// TIA Portal V17 export
// export: Created 2022-03-12T16:05:07.905036Z, ExportSetting WithDefaults, DisplayName Totally Integrated Automation Portal, DisplayVersion V17, DisplayName TIA Portal Openness, DisplayVersion V17, DisplayName TIA Portal Version Control Interface, DisplayVersion V17, DisplayName STEP 7 Professional, DisplayVersion V17, DisplayName STEP 7 Safety, DisplayVersion V17, DisplayName WinCC Advanced / Unified PC, DisplayVersion V17
ORGANIZATION_BLOCK "Main"   // OB1, LAD, ProgramCycle
TITLE = Main
{ S7_Optimized_Access := 'TRUE' }
AUTHOR : tech.team.motioncontrol@siemens.com
FAMILY : CPG
VERSION : 1.0
// Support: tech.team.motioncontrol@siemens.com
// Fax: +49 (0) 9131/98-1297
// stored: AutoNumber true, IsIECCheckEnabled false, SetENOAutomatically false
   VAR_INPUT
      Initial_Call : Bool;   // Initial call of this OB
      Remanence : Bool;   // =True, if remanent data are available
   END_VAR
   VAR_TEMP   // added for the SCL form of the ladder/FBD networks
      _w1 : Bool;
   END_VAR
BEGIN

REGION Network 1: Factory IO PLCSIM Communication
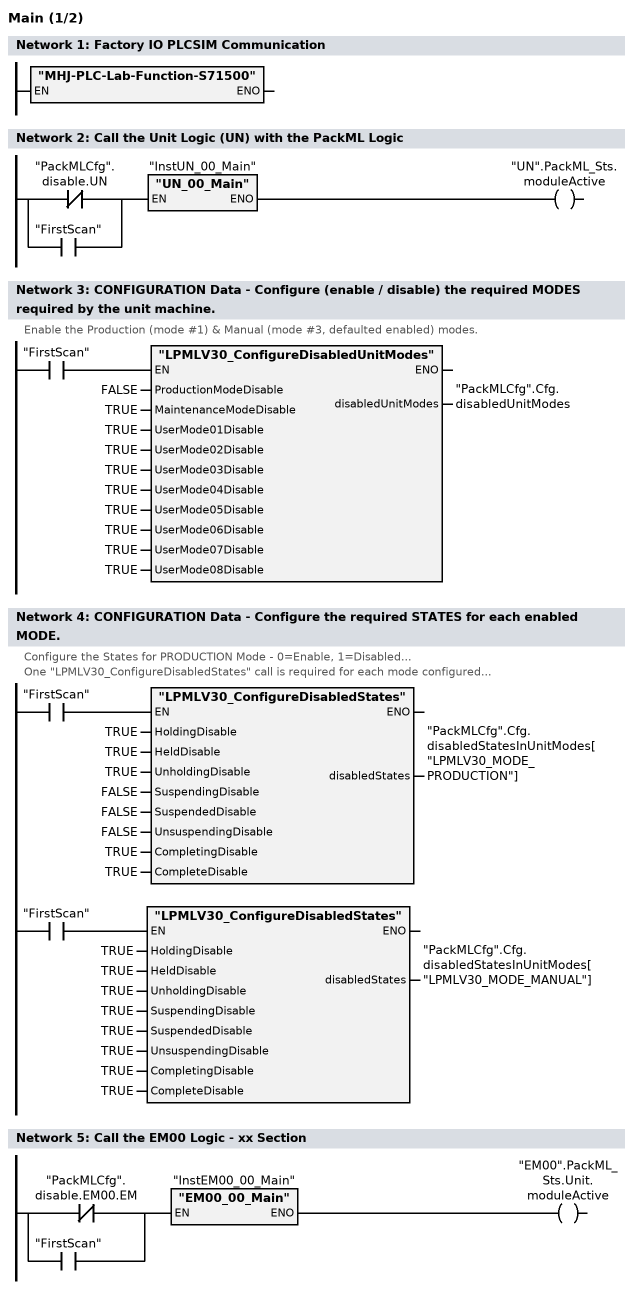
   RUNG wire#powerrail
      "MHJ-PLC-Lab-Function-S71500"()
   END_RUNG
   // the same network as SCL:
   "MHJ-PLC-Lab-Function-S71500"();
END_REGION

REGION Network 2: Call the Unit Logic (UN) with the PackML Logic
   RUNG wire#powerrail
      I_Contact( "PackMLCfg".disable.UN )
      wire#w1
      "InstUN_00_Main"()
      Coil( "UN".PackML_Sts.moduleActive )
   END_RUNG
   RUNG wire#powerrail
      Contact( "FirstScan" )
   END_RUNG wire#w1
   // the same network as SCL:
   "InstUN_00_Main"(EN := NOT "PackMLCfg".disable.UN OR "FirstScan", ENO => #_w1);   // "UN_00_Main"
   "UN".PackML_Sts.moduleActive := #_w1;
END_REGION

REGION Network 3: CONFIGURATION Data - Configure (enable / disable) the required MODES required by the unit machine.
   // Enable the Production (mode #1) & Manual (mode #3, defaulted enabled) modes.
   RUNG wire#powerrail
      Contact( "FirstScan" )
      "LPMLV30_ConfigureDisabledUnitModes"(ProductionModeDisable := FALSE, MaintenanceModeDisable := TRUE, UserMode01Disable := TRUE, UserMode02Disable := TRUE, UserMode03Disable := TRUE, UserMode04Disable := TRUE, UserMode05Disable := TRUE, UserMode06Disable := TRUE, UserMode07Disable := TRUE, UserMode08Disable := TRUE, disabledUnitModes => "PackMLCfg".Cfg.disabledUnitModes)
   END_RUNG
   // the same network as SCL:
   IF "FirstScan" THEN
       "LPMLV30_ConfigureDisabledUnitModes"(ProductionModeDisable := FALSE,
                               MaintenanceModeDisable := TRUE,
                               UserMode01Disable := TRUE,
                               UserMode02Disable := TRUE,
                               UserMode03Disable := TRUE,
                               UserMode04Disable := TRUE,
                               UserMode05Disable := TRUE,
                               UserMode06Disable := TRUE,
                               UserMode07Disable := TRUE,
                               UserMode08Disable := TRUE,
                               disabledUnitModes => "PackMLCfg".Cfg.disabledUnitModes);
   END_IF;
END_REGION

REGION Network 4: CONFIGURATION Data - Configure the required STATES for each enabled MODE.
   // Configure the States for PRODUCTION Mode - 0=Enable, 1=Disabled...
   // One "LPMLV30_ConfigureDisabledStates" call is required for each mode configured...
   RUNG wire#powerrail
      Contact( "FirstScan" )
      "LPMLV30_ConfigureDisabledStates"(HoldingDisable := TRUE, HeldDisable := TRUE, UnholdingDisable := TRUE, SuspendingDisable := FALSE, SuspendedDisable := FALSE, UnsuspendingDisable := FALSE, CompletingDisable := TRUE, CompleteDisable := TRUE, disabledStates => "PackMLCfg".Cfg.disabledStatesInUnitModes["LPMLV30_MODE_PRODUCTION"])
   END_RUNG
   RUNG wire#powerrail
      Contact( "FirstScan" )
      "LPMLV30_ConfigureDisabledStates"(HoldingDisable := TRUE, HeldDisable := TRUE, UnholdingDisable := TRUE, SuspendingDisable := TRUE, SuspendedDisable := TRUE, UnsuspendingDisable := TRUE, CompletingDisable := TRUE, CompleteDisable := TRUE, disabledStates => "PackMLCfg".Cfg.disabledStatesInUnitModes["LPMLV30_MODE_MANUAL"])
   END_RUNG
   // the same network as SCL:
   IF "FirstScan" THEN
       "LPMLV30_ConfigureDisabledStates"(HoldingDisable := TRUE,
                               HeldDisable := TRUE,
                               UnholdingDisable := TRUE,
                               SuspendingDisable := FALSE,
                               SuspendedDisable := FALSE,
                               UnsuspendingDisable := FALSE,
                               CompletingDisable := TRUE,
                               CompleteDisable := TRUE,
                               disabledStates => "PackMLCfg".Cfg.disabledStatesInUnitModes["LPMLV30_MODE_PRODUCTION"]);
   END_IF;
   IF "FirstScan" THEN
       "LPMLV30_ConfigureDisabledStates"(HoldingDisable := TRUE,
                               HeldDisable := TRUE,
                               UnholdingDisable := TRUE,
                               SuspendingDisable := TRUE,
                               SuspendedDisable := TRUE,
                               UnsuspendingDisable := TRUE,
                               CompletingDisable := TRUE,
                               CompleteDisable := TRUE,
                               disabledStates => "PackMLCfg".Cfg.disabledStatesInUnitModes["LPMLV30_MODE_MANUAL"]);
   END_IF;
END_REGION

REGION Network 5: Call the EM00 Logic - xx Section
   RUNG wire#powerrail
      I_Contact( "PackMLCfg".disable.EM00.EM )
      wire#w1
      "InstEM00_00_Main"()
      Coil( "EM00".PackML_Sts.Unit.moduleActive )
   END_RUNG
   RUNG wire#powerrail
      Contact( "FirstScan" )
   END_RUNG wire#w1
   // the same network as SCL:
   "InstEM00_00_Main"(EN := NOT "PackMLCfg".disable.EM00.EM OR "FirstScan", ENO => #_w1);   // "EM00_00_Main"
   "EM00".PackML_Sts.Unit.moduleActive := #_w1;
END_REGION

REGION Network 6: Call the EM01 Logic - xx Section
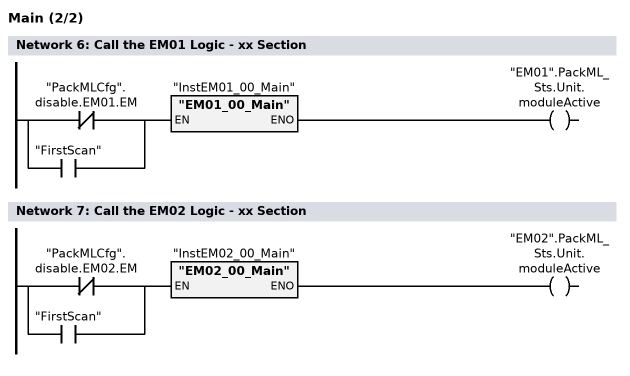
   RUNG wire#powerrail
      I_Contact( "PackMLCfg".disable.EM01.EM )
      wire#w1
      "InstEM01_00_Main"()
      Coil( "EM01".PackML_Sts.Unit.moduleActive )
   END_RUNG
   RUNG wire#powerrail
      Contact( "FirstScan" )
   END_RUNG wire#w1
   // the same network as SCL:
   "InstEM01_00_Main"(EN := NOT "PackMLCfg".disable.EM01.EM OR "FirstScan", ENO => #_w1);   // "EM01_00_Main"
   "EM01".PackML_Sts.Unit.moduleActive := #_w1;
END_REGION

REGION Network 7: Call the EM02 Logic - xx Section
   RUNG wire#powerrail
      I_Contact( "PackMLCfg".disable.EM02.EM )
      wire#w1
      "InstEM02_00_Main"()
      Coil( "EM02".PackML_Sts.Unit.moduleActive )
   END_RUNG
   RUNG wire#powerrail
      Contact( "FirstScan" )
   END_RUNG wire#w1
   // the same network as SCL:
   "InstEM02_00_Main"(EN := NOT "PackMLCfg".disable.EM02.EM OR "FirstScan", ENO => #_w1);   // "EM02_00_Main"
   "EM02".PackML_Sts.Unit.moduleActive := #_w1;
END_REGION
END_ORGANIZATION_BLOCK
